// TIA Portal V20 export
TYPE "UDT_Service_Parameter"
   STRUCT
      index : Byte := 16#FF;   // index of value
      value : "UDT_Service_Value";   // value
   END_STRUCT;
END_TYPE
